Staubli VAL3: page_instr.dtx

num nIndex
num nIndexItem = 1
num nKey = 255
public num nPage
num nRefresh = 2571.459
num nSelected
num nTime = 1
num nView
num nViewItem = 1
string sEvent = " 1 OUT valve1>ON"
string sField[2]
  [0] = "Disk://trajectory/PALLET/page_pallet"
  [1] = "hello"
public string sItems = "test"
string sList = " 1 OUT valve1>ON"
string sMenu[8]
  [2] = "I/O"
  [3] = "Paste"
  [4] = "Mark"
  [5] = "Delete"
  [6] = "Insert"
  [7] = "Save"
string sMenu8[8]
string sMessage
string sProgram = "test"
bool bButton[8]
  [1] = true
  [2] = true
  [3] = true
  [4] = true
  [5] = true
  [6] = true
  [7] = true
bool bExit = true
bool bLarge
num nId
bool bMoveRelease
num nOldIndex
string sPath
